RoboDK station: new_test.rdk

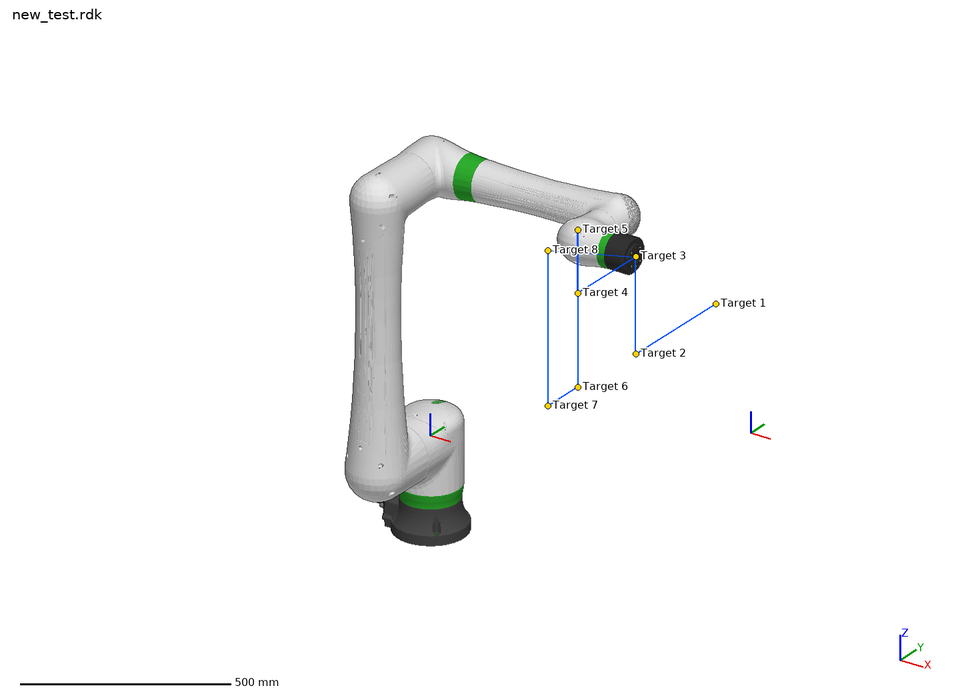
[picture v0: the station drawn from its stored meshes, robots at their saved joint values, targets as dots, program paths as lines]
Station new_test (saved by RoboDK 5.5.4). Poses are relative to the parent item; angles as X-Y-Z fixed-axis rotations.
Station parameters (name, value as stored): LIN64
  - frame Fanuc CRX-10iA/L Base at (0, 0, 245) mm
    - robot Fanuc CRX-10iA/L: 6 axes, payload 10 kg, reach 1418 mm, repeatability 0.05 mm, weight 40 kg
        modified DH rows (alpha deg, a mm, theta deg, d mm): 0, 0, 0, 245; -90, 0, -90, 0; 0, 710, 0, 0; -90, 0, 0, 540; 90, 0, 0, -150; -90, 0, 0, 160
        base shift (0, 0, -245) mm
        joint limits [-180, -180, -360, -190, -180, -190] to [180, 180, 430, 190, 180, 190]; home [0, 0, 0, 0, 0, 0]; saved at [0.006, 0.022, 1.828, 0.184, -1.828, -0.184]
  - frame Frame 2 at (1052.62, -177.96, 617) mm
    - target Target 1 (Cartesian target) at (-352.62, 359.73, 98.83) mm, rotated rx 0 ry -90 rz -180 deg; joints [24.333, 5.009, -10.679, -67.718, 26.441, 65.409] of Fanuc CRX-10iA/L
    - target Target 2 (Cartesian target) at (-352.62, 28.02, 98.83) mm, rotated rx 0 ry -90 rz -180 deg; joints [0.006, 4.426, -26.035, -0.014, 26.035, 0.012] of Fanuc CRX-10iA/L
    - target Target 3 (Cartesian target) at (-352.62, 28.02, 355.7) mm, rotated rx 0 ry -90 rz -180 deg; joints [0.006, 0.022, 1.828, 0.184, -1.828, -0.184] of Fanuc CRX-10iA/L
    - target Target 4 (Cartesian target) at (-352.62, -211.77, 355.7) mm, rotated rx 0 ry -90 rz 180 deg; joints [-30.093, 8.646, 16.639, -63.706, -34.005, 59.204] of Fanuc CRX-10iA/L
    - target Target 5 (Cartesian target) at (-352.62, -211.77, 522.54) mm, rotated rx 0 ry -90 rz 180 deg; joints [-26.345, 11.76, 32.014, -43.05, -40.549, 35.367] of Fanuc CRX-10iA/L
    - target Target 6 (Cartesian target) at (-352.62, -211.77, 107.3) mm, rotated rx 0 ry -90 rz 180 deg; joints [-37.884, 12.073, -7.245, -99.207, -38.469, 101.697] of Fanuc CRX-10iA/L
    - target Target 7 (Cartesian target) at (-352.62, -334.41, 107.3) mm, rotated rx 0 ry -90 rz 180 deg; joints [-44.517, 17.997, -5.005, -95.07, -44.738, 97.12] of Fanuc CRX-10iA/L
    - target Target 8 (Cartesian target) at (-352.62, -334.41, 517.51) mm, rotated rx 0 ry -90 rz 180 deg; joints [-36.317, 18.963, 35.529, -51.67, -49.024, 39.673] of Fanuc CRX-10iA/L
    - target Target 3 (Cartesian target) at (-352.62, 28.02, 355.7) mm, rotated rx 0 ry -90 rz -180 deg; joints [0.006, 0.022, 1.828, 0.184, -1.828, -0.184] of Fanuc CRX-10iA/L
  - Python program testCRX10Model_10 (listed below)
  - Python program Prog2 (listed below)
  - program Prog3 (10 instructions, listed below)
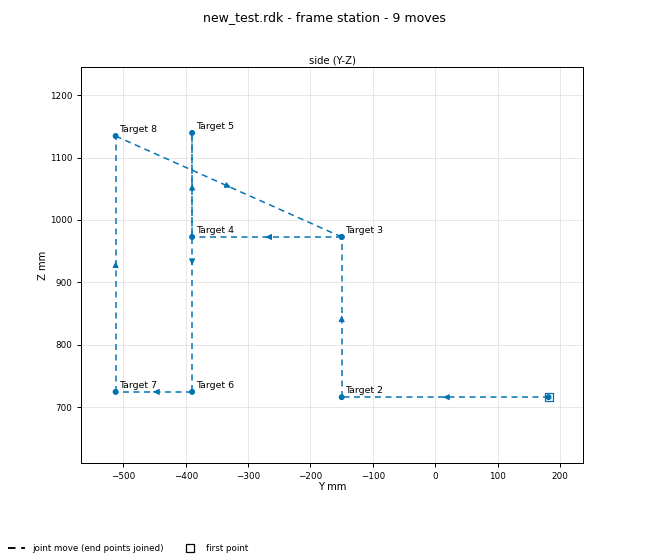
[picture p0: tool path of new_test.rdk in frame station, 9 of 9 moves have a stored position in this frame; points joined in program order, loops and branches not executed]

--- Python program testCRX10Model_10 ---
import time

from robodk.robolink import *                  # import the robolink library
RDK = Robolink()                        # connect to the RoboDK API (RoboDK starts if it has not started

robots = RDK.ItemList(ITEM_TYPE_ROBOT)
print(robots)


# tool  = RDK.Item('SCHUNK- 1321170 Co-act EGP-C 40-N-N-KTOE_ 0')                # Get an item named Tool (name in the RoboDK station tree)

robot = RDK.Item('', ITEM_TYPE_ROBOT)   # Get the first available robot


robot.Connect()
RDK.setRunMode(RUNMODE_RUN_ROBOT)
#RDK.setRunMode(RUNMODE_SIMULATE)
#frame = RDK.ItemUserPick('Select a reference frame', ITEM_TYPE_FRAME)   # Promt the user to select a reference frame
frame = RDK.Item('Frame 2', ITEM_TYPE_FRAME)

robot.setPoseFrame(frame)
# robot.setPoseTool(tool)

robot.setSpeed(1500)

for i in range(0,1):
	print("Run: ", i)
	# use set speed at the start and inbetween movements.
	# for move joint use speed_joints and set a float value (based on degs/sec^2)
	robot.setSpeed(1500, speed_joints = 5)
	target = RDK.Item('Target 1', ITEM_TYPE_TARGET)   # Get a target called "turn1"
	robot.MoveJ(target)             # Move the robot to the target using the selected reference frame
	robot.setSpeed(3000, speed_joints = 5)
	# time.sleep(1.0)
	robot.setSpeed(500, speed_joints = 5)
	target = RDK.Item('Target 2', ITEM_TYPE_TARGET)   # Get a target called "home"
	robot.MoveJ(target)             # Move the robot to the target using the selected reference frame
	robot.setSpeed(3000, speed_joints = 50)


	#target = RDK.Item('Turn3', ITEM_TYPE_TARGET)   # Get a target called "home"
	#kjjrobot.MoveJ(target)             # Move the robot to the target using the selected reference frame



	target = RDK.Item('Target 3', ITEM_TYPE_TARGET)   # Get a target called "home"
	robot.MoveJ(target)             # Move the robot to the target using the selected reference frame
	robot.setSpeed(3000, speed_joints = 50)

	target = RDK.Item('Target 4', ITEM_TYPE_TARGET)   # Get a target called "home"
	robot.MoveJ(target)             # Move the robot to the target using the selected reference frame
	robot.setSpeed(3000, speed_joints = 30)
	target = RDK.Item('Target 5', ITEM_TYPE_TARGET)   # Get a target called "home"
	robot.MoveJ(target)             # Move the robot to the target using the selected reference frame
	robot.setSpeed(3000, speed_joints = 40)
	target = RDK.Item('Target 6', ITEM_TYPE_TARGET)   # Get a target called "home"
	robot.MoveJ(target)             # Move the robot to the target using the selected reference frame
	robot.setSpeed(3000, speed_joints = 50)
	target = RDK.Item('Target 7', ITEM_TYPE_TARGET)   # Get a target called "home"
	robot.MoveJ(target)             # Move the robot to the target using the selected reference frame
	robot.setSpeed(3000, speed_joints = 60)
	target = RDK.Item('Target 8', ITEM_TYPE_TARGET)   # Get a target called "home"
	robot.MoveJ(target)             # Move the robot to the target using the selected reference frame

	target = RDK.Item('Target 3', ITEM_TYPE_TARGET)   # Get a target called "home"
	robot.MoveJ(target)             # Move the robot to the target using the selected reference frame

--- Python program Prog2 ---
# Type help("robodk.robolink") or help("robodk.robomath") for more information
# Press F5 to run the script
# Documentation: https://robodk.com/doc/en/RoboDK-API.html
# Reference:     https://robodk.com/doc/en/PythonAPI/robodk.html
# Note: It is not required to keep a copy of this file, your Python script is saved with your RDK project

# You can also use the new version of the API:
from robodk import robolink    # RoboDK API
from robodk import robomath    # Robot toolbox
RDK = robolink.Robolink()

# Forward and backwards compatible use of the RoboDK API:
# Remove these 2 lines to follow python programming guidelines
from robodk import *      # RoboDK API
from robolink import *    # Robot toolbox
# Link to RoboDK
# RDK = Robolink()

# Notify user:
print('To edit this program:\nright click on the Python program, then, select "Edit Python script"')

# Program example:
item = RDK.Item('base')
if item.Valid():
    print('Item selected: ' + item.Name())
    print('Item posistion: ' + repr(item.Pose()))

print('Items in the station:')
itemlist = RDK.ItemList()
print(itemlist)

# Provoking an exception will display the console output if you run this script from RoboDK
raise Exception('Program not edited.')

--- program Prog3 (robot Fanuc CRX-10iA/L) ---
  Set Ref.: Frame 2
  MoveJ (Target 1)
  MoveJ (Target 2)
  MoveJ (Target 3)
  MoveJ (Target 4)
  MoveJ (Target 5)
  MoveJ (Target 6)
  MoveJ (Target 7)
  MoveJ (Target 8)
  MoveJ (Target 3)
